PROGRAM Arrays

END_PROGRAM

(* stored: Version 1.1.0.1
   POU Arrays: Id {cbc8e7a1-469d-4f0b-975e-c0483b44ad8c}, SpecialFunc None *)
